TYPE InputBase_8311D824 :
STRUCT
END_STRUCT
END_TYPE

(* stored: Version 1.2.0.0, ProductVersion 3.1.4024.9
   DUT InputBase_8311D824: Id {8c9590e7-e6b4-4f80-9517-14c3b6bb67da} *)
